FUNCTION_BLOCK AutoResetCdt_HMI (* Service Interface Function Block Type *)
  (* Standard: 61499-2 *)
  (* Version 0.0, 8/3/2026, Schneider Electric, template *)
  PACKAGE SE.Nereda;
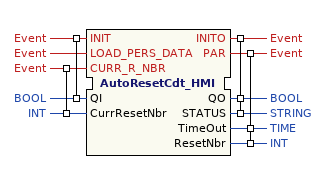
  EVENT_INPUT
    INIT WITH QI;
    LOAD_PERS_DATA;
    CURR_R_NBR WITH CurrResetNbr;
  END_EVENT
  EVENT_OUTPUT
    INITO WITH QO, STATUS;
    PAR WITH TimeOut, ResetNbr;
  END_EVENT
  VAR_INPUT
    QI : BOOL;
    CurrResetNbr : INT;
  END_VAR
  VAR_OUTPUT
    QO : BOOL; (* Event Output Qualifier *)
    STATUS : STRING; (* Service Status *)
    TimeOut : TIME;
    ResetNbr : INT;
  END_VAR
  SERVICE /
    SEQUENCE 
    END_SEQUENCE
  END_SERVICE
END_FUNCTION_BLOCK
